FUNCTION_BLOCK FB_ChannelReset

VAR_INPUT
	i_Reset:BOOL;
	i_ChannelID: UDINT;

END_VAR
VAR_OUTPUT
END_VAR
VAR
	fbReset: ItpReset;
END_VAR

fbReset(
	bExecute:= i_Reset,
	nChnId:= i_ChannelID,
	tTimeOut:= T#1S,
	bBusy=> ,
	bErr=> ,
	nErrId=> );

END_FUNCTION_BLOCK

(* stored: Version 1.1.0.1, ProductVersion 3.1.4024.10
   POU FB_ChannelReset: Id {48ca0b5c-dde0-460d-a003-088c45c13a7a}, SpecialFunc None *)
